FUNCTION_BLOCK NeredaEffluent (* CAT Function Block Type *)
  (* Standard: 61499-2 *)
  (* Version 0.0, 6/13/2026, Schneider Electric, template *)
  PACKAGE SE.Nereda;
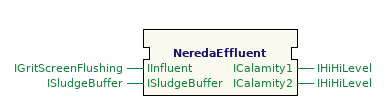
  SOCKETS
    IInfluent : IGritScreenFlushing;
    ISludgeBuffer : ISludgeBuffer;
  END_SOCKETS
  PLUGS
    ICalamity1 : IHiHiLevel;
    ICalamity2 : IHiHiLevel;
  END_PLUGS
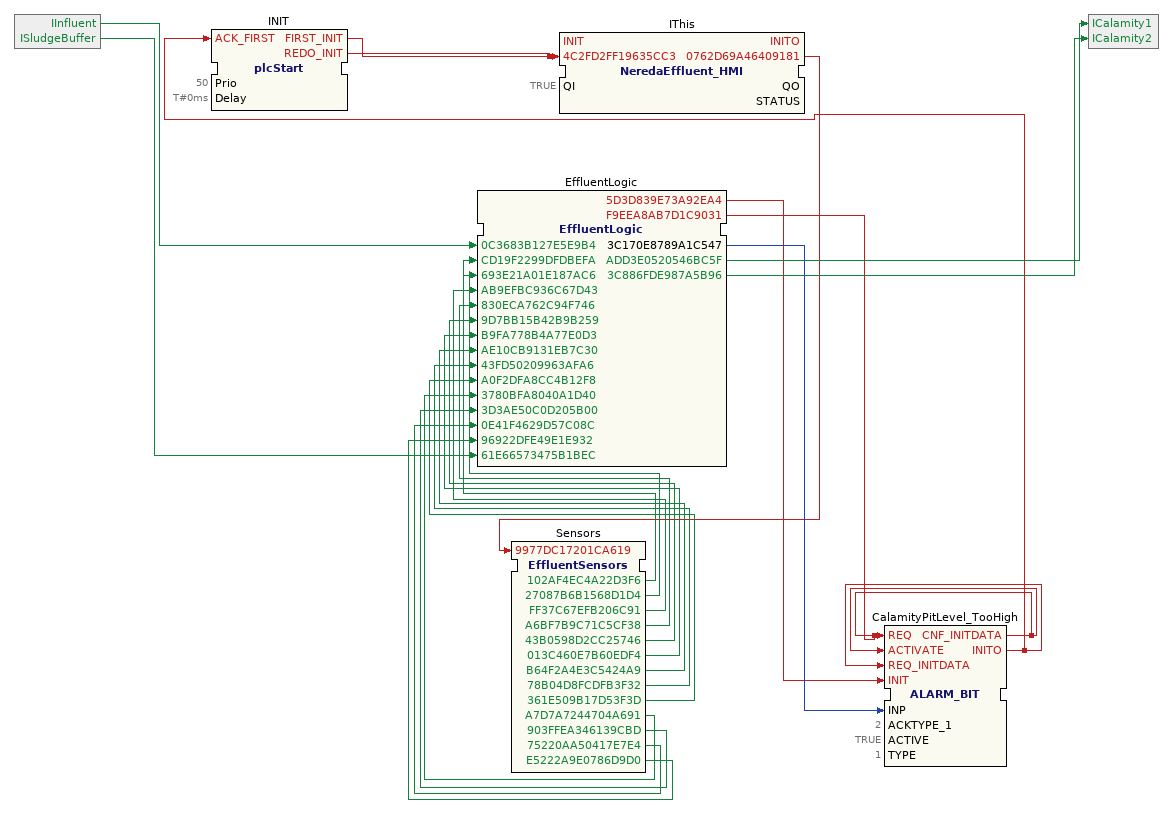
  (* 01 - FUNCTIONNAL INPUT INTERFACE *)
  (* 00 - INITIALIZATION *)
  (* 05 - LOGIC *)
  (* 06 - HMI INTERFACE *)
  (* 03 - FIELD INTERFACE *)
  (* 02 - FUNCTIONNAL OUTPUT INTERFACE *)
  (* Effluent Logic *)
  (* 04 - CHILDREN *)
  (* 4A - TYPICALS *)
  (* ALARMS - Calamity *)
  FBS
    INIT : plcStart(Prio := 50, Delay := T#0ms);
    IThis : NeredaEffluent_HMI(QI := TRUE);
    EffluentLogic : EffluentLogic;
    Sensors : EffluentSensors;
    CalamityPitLevel_TooHigh : ALARM_BIT(ACKTYPE_1 := 2, ACTIVE := TRUE, TYPE := 1);
  END_FBS
  EVENT_CONNECTIONS
    INIT.FIRST_INIT TO IThis.4C2FD2FF19635CC3;
    INIT.REDO_INIT TO IThis.4C2FD2FF19635CC3;
    CalamityPitLevel_TooHigh.CNF_INITDATA TO CalamityPitLevel_TooHigh.REQ;
    CalamityPitLevel_TooHigh.CNF_INITDATA TO CalamityPitLevel_TooHigh.ACTIVATE;
    CalamityPitLevel_TooHigh.INITO TO CalamityPitLevel_TooHigh.REQ_INITDATA;
    CalamityPitLevel_TooHigh.INITO TO INIT.ACK_FIRST;
    EffluentLogic.5D3D839E73A92EA4 TO CalamityPitLevel_TooHigh.INIT;
    EffluentLogic.F9EEA8AB7D1C9031 TO CalamityPitLevel_TooHigh.REQ;
    IThis.0762D69A46409181 TO Sensors.9977DC17201CA619;
  END_CONNECTIONS
  DATA_CONNECTIONS
    EffluentLogic.3C170E8789A1C547 TO CalamityPitLevel_TooHigh.INP;
  END_CONNECTIONS
  ADAPTER_CONNECTIONS
    IInfluent TO EffluentLogic.0C3683B127E5E9B4;
    Sensors.102AF4EC4A22D3F6 TO EffluentLogic.CD19F2299DFDBEFA;
    Sensors.27087B6B1568D1D4 TO EffluentLogic.693E21A01E187AC6;
    Sensors.FF37C67EFB206C91 TO EffluentLogic.AB9EFBC936C67D43;
    Sensors.A6BF7B9C71C5CF38 TO EffluentLogic.830ECA762C94F746;
    Sensors.43B0598D2CC25746 TO EffluentLogic.9D7BB15B42B9B259;
    Sensors.013C460E7B60EDF4 TO EffluentLogic.B9FA778B4A77E0D3;
    Sensors.B64F2A4E3C5424A9 TO EffluentLogic.AE10CB9131EB7C30;
    Sensors.78B04D8FCDFB3F32 TO EffluentLogic.43FD50209963AFA6;
    Sensors.361E509B17D53F3D TO EffluentLogic.A0F2DFA8CC4B12F8;
    Sensors.A7D7A7244704A691 TO EffluentLogic.3780BFA8040A1D40;
    Sensors.903FFEA346139CBD TO EffluentLogic.3D3AE50C0D205B00;
    Sensors.75220AA50417E7E4 TO EffluentLogic.0E41F4629D57C08C;
    Sensors.E5222A9E0786D9D0 TO EffluentLogic.96922DFE49E1E932;
    ISludgeBuffer TO EffluentLogic.61E66573475B1BEC;
    EffluentLogic.ADD3E0520546BC5F TO ICalamity1;
    EffluentLogic.3C886FDE987A5B96 TO ICalamity2;
  END_CONNECTIONS
END_FUNCTION_BLOCK
